VAR_INST
	//This error cannot be reset. Requires a reset cold
	{attribute 'hide'}	
	fbInitError : FB_TcAlarm;
END_VAR
// Check if link to track is mapped
IF NOT THIS^.Mapped THEN
	IF NOT fbInitError.bRaised THEN 
		//This error cannot be reset. Requires a reset cold
		fbInitError.CreateEx(stEventEntry:=TC_EVENTS.CHALET_Base_Events.VariableLinkMissing, ipSourceInfo := THIS^.fbSourceInfo, bWithConfirmation := FALSE);
		stVarInfo := __VARINFO(THIS^.fbTrack.MCTOPLC_STD);
		fbInitError.ipArguments.AddString(stVarInfo.Symbol);
		fbInitError.Raise(0);
	END_IF
	Initialize := E_FAIL;
	RETURN;
END_IF


IF NOT bInitDone THEN
	//Busy
	Initialize := S_PENDING;
	
	
	//TRUE = Use inside PLC the track name from the TcCom Track Object. 
	//FALSE = overwride TcCom Track object with instance name
	FW_ObjMgr_GetObjectInstance(oid:= THIS^.fbTrack.MCTOPLC_STD.TrackOID, iid:= TC_GLOBAL_IID_LIST.IID_ITComObject, pipUnk:= ADR(pObject));
	IF XPlanarParameterlist.B_TRACK_NAME_TACKOVER_FROM_TRACK_OBJECT THEN
		IF pObject <> 0 THEN
			pObject.TcGetObjectName(objName:= ADR(sName), nameLen := SIZEOF(sName));
			pObject.TcRelease();
			THIS^.fbSourceInfo.sName := sName;
		END_IF
	ELSE
		IF pObject <> 0 THEN
			sName := THIS^.LUID;
			pObject.TcSetObjectName(ADR(sName));
			pObject.TcRelease();
		END_IF
	END_IF

	
	//Done as sone list is initilized
	bInitDone := TRUE;
	
ELSE	
	//Done
	Initialize := S_OK;	
END_IF



THIS^.fbFeedback.ActiveCommand 		:= TO_STRING(CHALET_NC.E_NcAxisCommands.Initialize);
THIS^.eActiveCommand 				:= CHALET_NC.E_NcAxisCommands.Initialize;
THIS^.fbFeedback.LastCommandAccepted:= TRUE;	
//Set done or keep in busy state	
THIS^.fbFeedback.HR := Initialize;
END_METHOD

{attribute 'monitoring':='call'}
//[mm]
PROPERTY Length : LREAL
GET
Length := THIS^.fbTrack.GetLength();
END_GET
END_PROPERTY

{attribute 'monitoring':='call'}
PROPERTY Mapped : BOOL //Project is mapped to MC (McToPlc and PlcToMc)
GET
VAR
	bMcToPlcNotMapped 	: BOOL;
END_VAR
bMcToPlcNotMapped := F_GetMappingStatus(ADR(THIS^.fbTrack.MCTOPLC_STD), SIZEOF(THIS^.fbTrack.MCTOPLC_STD)) <> EPlcMappingStatus.MS_Mapped;

Mapped := NOT bMcToPlcNotMapped;
END_GET
END_PROPERTY

{attribute 'monitoring':='call'}
//List of interfaces to movers on this track
PROPERTY MoversOnTrack : I_CH_LIST
GET
THIS^.Prepare();//Prepare a list movers on this track


MoversOnTrack := THIS^.fbListOfMoversOnTrack;
END_GET
END_PROPERTY

{attribute 'monitoring':='call'}
//Unique object ID
PROPERTY OID : OTCID
GET
OID := THIS^.fbTrack.MCTOPLC_STD.TrackOID;
END_GET
END_PROPERTY

{attribute 'monitoring':='call'}
//List of interfaces to paths on this track
PROPERTY PathsOnTrack : I_CH_List
GET
THIS^.Prepare();//Prepare a list stations on this track

PathsOnTrack := THIS^.fbListPathsOnThisTrack;
END_GET
END_PROPERTY

{attribute 'monitoring':='call'}
PROPERTY PlanarTrack : REFERENCE TO MC_PlanarTrack
GET
PlanarTrack ref= THIS^.fbTrack;
END_GET
END_PROPERTY

(* Time-critical information is processed here, which can then be polled via the property every cycle. 
The update method is usually at the end of the program and then it is already 'outdated'. *)
METHOD PRIVATE Prepare : HRESULT
VAR
	ipThisTrack : I_XP_Track := THIS^;
	ipStation : I_XP_Station;
	ipMover : I_XP_Mover;
	ipPath : I_XP_Path;

END_VAR

VAR_INST
	{attribute 'hide'}
	nLastUpdatedCycleCount : UDINT;
END_VAR
//Check if this Cycle the dates are allready prepared
IF nLastUpdatedCycleCount <> TwinCAT_SystemInfoVarList._TaskInfo[THIS^.nTaskIndex].CycleCount THEN
	nLastUpdatedCycleCount := TwinCAT_SystemInfoVarList._TaskInfo[THIS^.nTaskIndex].CycleCount;

	//Creat a list of all Stations on this Track
	THIS^.fbListOfStationsOnTrack.Clear();
	THIS^.ipXpSystem.Stations.ResetIterator();
	WHILE THIS^.ipXpSystem.Stations.HasNextObject() DO
		IF ToXpStation(THIS^.ipXpSystem.Stations.GetNextObject(), ipStation) AND_THEN ipStation.AccocietedTrack <> 0 AND_THEN ipStation.AccocietedTrack = ipThisTrack THEN
			THIS^.fbListOfStationsOnTrack.AddObject(ipStation);
		END_IF
	END_WHILE
	THIS^.ipXpSystem.Stations.RestoreIterator();
	
	
	
	//Creat a list of all Movers on this Track
	THIS^.fbListOfMoversOnTrack.Clear();
	THIS^.ipXpSystem.Movers.ResetIterator();
	WHILE THIS^.ipXpSystem.Movers.HasNextObject() DO
		IF ToXpMover(THIS^.ipXpSystem.Movers.GetNextObject(), ipMover) AND_THEN ipMover.CurrentTrack <> 0 AND_THEN ipMover.CurrentTrack = ipThisTrack THEN
			THIS^.fbListOfMoversOnTrack.AddObject(ipStation);
		END_IF
	END_WHILE
	THIS^.ipXpSystem.Movers.RestoreIterator();	
	
	
		
	//Creat a list of all Paths on this Track
	THIS^.fbListPathsOnThisTrack.Clear();
	THIS^.ipXpSystem.Paths.ResetIterator();
	WHILE THIS^.ipXpSystem.Paths.HasNextObject() DO
		IF __QUERYINTERFACE(THIS^.ipXpSystem.Paths.GetNextObject(), ipPath)AND_THEN __ISVALIDREF(ipPath.TracksUsed) AND_THEN ipPath.TracksUsed.ObjectInList(ipThisTrack) THEN
			THIS^.fbListPathsOnThisTrack.AddObject(ipPath);
		END_IF
	END_WHILE
	THIS^.ipXpSystem.Paths.RestoreIterator();	
	
END_IF
END_METHOD

METHOD Reset : HRESULT
VAR_INPUT
END_VAR
THIS^.eActiveCommand 				:= CHALET_NC.E_NcAxisCommands.Reset;
THIS^.fbFeedback.LastCommandAccepted:= TRUE;		
THIS^.fbFeedback.Busy 				:= TRUE;

THIS^.fbTrack.Reset(THIS^.fbFeedbackReset);
Reset := S_OK;
END_METHOD

(* Returns the first station on current track who has exact thsi position or is ahead
	If no station on this track, result is maybe on another track*)
METHOD StationAhedPosition : I_XP_Station
VAR_INPUT
	fPosOnTrack : LREAL;//[mm]	
END_VAR
VAR
	fDistToTempBestStaton : LREAL := CHALET_BaseComponents.GVL_Datatypes.cMaxLreal;;
	ipTempBestStation : I_XP_Station;
	fDist :LREAL;
	bStartAndEndIsOnThisTrack : BOOL;
	ipThisTrack : I_XP_Track := (THIS^);
	ipEachPathOnTrack : I_XP_Path;
END_VAR
THIS^.fbListPathsOnThisTrack.ResetIterator();
WHILE THIS^.fbListPathsOnThisTrack.HasNextObject() DO
	IF __QUERYINTERFACE(THIS^.fbListPathsOnThisTrack.GetNextObject(), ipEachPathOnTrack) THEN
		
		bStartAndEndIsOnThisTrack := ipEachPathOnTrack.StationStart.AccocietedTrack = ipThisTrack AND ipEachPathOnTrack.StationDestination.AccocietedTrack = ipThisTrack; 
		
		//Check if end of route is not before this station
		IF (ipEachPathOnTrack.StationDestination.AccocietedTrack = ipThisTrack) AND (ipEachPathOnTrack.StationDestination.PositionOnTrack < fPosOnTrack) AND NOT bStartAndEndIsOnThisTrack THEN
			//end is before the searched position - not a valide targed
			CONTINUE;		
		END_IF
		
		//Check if end of route is before this station - CLOSED LOOP, SHORT SEGMENT
		IF NOT F_InLimitTest(fMinimum := ipEachPathOnTrack.StationStart.PositionOnTrack, fInput:= fPosOnTrack, fMaximum := ipEachPathOnTrack.StationDestination.PositionOnTrack) AND bStartAndEndIsOnThisTrack THEN
			//end is before the searched position - not a valide targed
			CONTINUE;		
		END_IF
	
			
		fDist := ipEachPathOnTrack.DistanceToDestiantion(	ipTrack := ipThisTrack, 
															fPosOnTrack := 	fPosOnTrack);
															
		//Get shortest distance													
		IF 	fDist <= fDistToTempBestStaton	THEN
			fDistToTempBestStaton := fDist;
			ipTempBestStation := ipEachPathOnTrack.StationDestination;
		END_IF
		
	END_IF
END_WHILE
THIS^.fbListPathsOnThisTrack.RestoreIterator();

StationAhedPosition := ipTempBestStation;
END_METHOD

{attribute 'monitoring':='call'}
//List of interfaces to stations on this track
PROPERTY StationsOnTrack : I_CH_List
GET
THIS^.Prepare();//Prepare a list stations on this track

StationsOnTrack := THIS^.fbListOfStationsOnTrack;
END_GET
END_PROPERTY

{attribute 'monitoring':='call'}
//List of interfaces from other tracks
PROPERTY TracksAhead : I_CH_List
GET
TracksAhead := fbTracksAhead;
END_GET
END_PROPERTY

{attribute 'monitoring':='call'}
//List of interfaces from other tracks
PROPERTY TracksBehinde : I_CH_List
GET
TracksBehinde:= fbTracksBehinde;
END_GET
END_PROPERTY

{attribute 'monitoring':='call'}
//zzz Todo Delet me
PROPERTY TracksEndAtThis : REFERENCE TO  ARRAY[0..(XPlanarParameterlist.N_MAX_STATIONS_AHEAD_OR_BEHIND-1)] OF I_XP_Track
GET
TracksEndAtThis REF= ipTracksEndAtThis;
END_GET
END_PROPERTY

{attribute 'monitoring':='call'}
PROPERTY TracksStartFromThis : REFERENCE TO ARRAY[0..(XPlanarParameterlist.N_MAX_STATIONS_AHEAD_OR_BEHIND-1)] OF I_XP_Track
GET
TracksStartFromThis REF= ipTracksStartFromThis;
END_GET
END_PROPERTY

METHOD PUBLIC Update : HRESULT
VAR_INPUT
END_VAR

THIS^.Prepare();//Prepare time-critical information, if not already done



// ********************** Set feedback depending on active command *******************************
IF THIS^.eActiveCommand <> E_NcAxisCommands.None THEN
	fbFeedback.ActiveCommand 	:= TO_STRING(THIS^.eActiveCommand);	
END_IF

CASE THIS^.eActiveCommand OF
	E_NcAxisCommands.None: 
		//Display if a Mover Error is active during no command is active
		IF THIS^.fbTrack.Error AND NOT fbFeedback.Error THEN 
			fbFeedback.ErrorId 			:= THIS^.fbTrack.ErrorID;
			fbFeedback.ActiveCommand 	:= TO_STRING(E_NcAxisCommands.None);	
			fbFeedback.ClearObjectInfo();
		END_IF

	E_NcAxisCommands.Initialize:
		fbFeedback.Busy 			:= NOT THIS^.bInitDone;
		fbFeedback.Done 			:= THIS^.bInitDone;
		fbFeedback.ErrorId 			:= 0;
		fbFeedback.ClearObjectInfo();
		                        	
	E_NcAxisCommands.Enable:     	
		fbFeedback.Busy 			:= fbFeedbackEnable.Busy;
		fbFeedback.Done 			:= fbFeedbackEnable.Done;
		fbFeedback.ErrorId 			:= fbFeedbackEnable.ErrorID;
        fbFeedback.ObjectInfo		:= fbFeedbackEnable.objectInfo;
                                			                        	
	E_NcAxisCommands.Disable:     	
		fbFeedback.Busy 			:= fbFeedbackDisable.Busy;
		fbFeedback.Done 			:= fbFeedbackDisable.Done;
		fbFeedback.ErrorId 			:= fbFeedbackDisable.ErrorID;
        fbFeedback.ObjectInfo		:= fbFeedbackDisable.objectInfo;
		
	E_NcAxisCommands.Configure:
		fbFeedback.Busy 		:= nSeqConfiguring > 0;
		fbFeedback.Done 		:= nSeqConfiguring = 999;
		IF nSeqConfiguring > 1000 THEN
			fbFeedback.ErrorId 		:= nSeqConfiguring;
		END_IF
                                			                        	
	E_NcAxisCommands.Reset:     	
		fbFeedback.Busy 			:= fbFeedbackReset.Busy;
		fbFeedback.Done 			:= fbFeedbackReset.Done;
		fbFeedback.ErrorId 			:= fbFeedbackReset.ErrorID;
        fbFeedback.ObjectInfo		:= fbFeedbackReset.objectInfo;
                                      			                        	
	E_NcAxisCommands.AddToGroupe:     	
		fbFeedback.Busy 			:= fbFeedbackAddToGrp.Busy;
		fbFeedback.Done 			:= fbFeedbackAddToGrp.Done;
		fbFeedback.ErrorId 			:= fbFeedbackAddToGrp.ErrorID;
        fbFeedback.ObjectInfo		:= fbFeedbackAddToGrp.objectInfo;
                                      			                        	
	E_NcAxisCommands.RemoveFromGroupe:     	
		fbFeedback.Busy 			:= fbFeedbackRmvFromGrp.Busy;
		fbFeedback.Done 			:= fbFeedbackRmvFromGrp.Done;
		fbFeedback.ErrorId 			:= fbFeedbackRmvFromGrp.ErrorID;
        fbFeedback.ObjectInfo		:= fbFeedbackRmvFromGrp.objectInfo;
                                		
	ELSE//External command in subclass
		;
END_CASE


// **********************  Stop to execute commands on .done or .error ***************************
IF fbFeedback.Done OR THIS^.fbFeedback.Error THEN
	eActiveCommand 				:= E_NcAxisCommands.None;
END_IF

//Update xplanar object
THIS^.fbTrack.Update();

//Update feedback object
fbFeedbackEnable.Update(); 
fbFeedbackDisable.Update(); 
fbFeedbackReset.Update(); 
fbFeedbackAddToGrp.Update(); 
fbFeedbackRmvFromGrp.Update();
END_METHOD

END_FUNCTION_BLOCK

// FUNCTIONs/F_InLimitTest
FUNCTION F_InLimitTest : BOOL
VAR_INPUT
	fMinimum 	: LREAL;
	fMaximum 	: LREAL;
	fInput 		: LREAL;
END_VAR

//Normal case
// 9 Max
// 5 Test
// 1 Min
IF fMinimum <= fMaximum THEN
	F_InLimitTest := (fInput >= fMinimum) AND (fInput <= fMaximum);
	
//Modulo case	
// 6 | 6  Max
// 5 | 9  Test
// 8 | 8  Min
ELSIF fMinimum > fMaximum THEN
	F_InLimitTest := NOT((fInput > fMaximum) AND (fInput < fMinimum));
END_IF

END_FUNCTION

// COMPONENTs/Track/I_XP_Track_PLC
INTERFACE I_XP_Track_PLC EXTENDS I_CH_Object

{attribute 'monitoring':='call'}
PROPERTY CtsMoversOnTrack : UINT
GET
END_GET
END_PROPERTY

{attribute 'monitoring':='call'}
PROPERTY Feedback : I_XP_Feedback
GET
END_GET
END_PROPERTY

{attribute 'monitoring':='call'}
//[mm]
PROPERTY Length : LREAL
GET
END_GET
END_PROPERTY

{attribute 'monitoring':='call'}
PROPERTY Mapped : BOOL //Project is mapped to MC (McToPlc and PlcToMc)
GET
END_GET
END_PROPERTY

{attribute 'monitoring':='call'}
//Unique object ID
PROPERTY OID : OTCID
GET
END_GET
END_PROPERTY

{attribute 'monitoring':='call'}
PROPERTY PlanarTrack : REFERENCE TO MC_PlanarTrack
GET
END_GET
END_PROPERTY

(* Returns the first station on current track who has exact thsi position or is ahead
	If no station on this track, result is maybe on another track*)
METHOD StationAhedPosition : I_XP_Station
VAR_INPUT
	fPosOnTrack : LREAL;//[mm]	
END_VAR
END_METHOD

{attribute 'monitoring':='call'}
//List of interfaces to stations on this track
PROPERTY StationsOnTrack : I_CH_List
GET
END_GET
END_PROPERTY

{attribute 'monitoring':='call'}
//List of interfaces from other tracks
PROPERTY TracksAhead : I_CH_List
GET
END_GET
END_PROPERTY

{attribute 'monitoring':='call'}
//List of interfaces from other tracks
PROPERTY TracksBehinde : I_CH_List
GET
END_GET
END_PROPERTY

{attribute 'monitoring':='call'}
PROPERTY TracksEndAtThis : REFERENCE TO  ARRAY[0..(XPlanarParameterlist.N_MAX_STATIONS_AHEAD_OR_BEHIND-1)] OF I_XP_Track
GET
END_GET
END_PROPERTY

{attribute 'monitoring':='call'}
PROPERTY TracksStartFromThis : REFERENCE TO ARRAY[0..(XPlanarParameterlist.N_MAX_STATIONS_AHEAD_OR_BEHIND-1)] OF I_XP_Track
GET
END_GET
END_PROPERTY

END_INTERFACE
